{attribute 'linkalways'} 
{attribute 'no_explicit_call' := 'This FB is a CLASS and must be accessed using methods or properties'}
{attribute 'enable_dynamic_creation'}
FUNCTION_BLOCK Node_ContainerType_Vector_TcVnVector4_REAL EXTENDS Node
VAR
    out : _GUID;
END_VAR

METHOD PUBLIC  Clone : I_Node
VAR
	pNode : POINTER TO Node_ContainerType_Vector_TcVnVector4_REAL;
END_VAR
pNode := __NEW(Node_ContainerType_Vector_TcVnVector4_REAL);
Clone := pNode^;
END_METHOD

METHOD FB_init : BOOL
VAR_INPUT
	bInitRetains : BOOL; // if TRUE, the retain variables are initialized (warm start / cold start)
	bInCopyCode : BOOL;  // if TRUE, the instance afterwards gets moved into the copy code (online change)
END_VAR
AddOutput('out', out);
END_METHOD

METHOD PROTECTED OnExecute
out.Value := ContainerType_Vector_TcVnVector4_REAL;
END_METHOD

END_FUNCTION_BLOCK

(* stored: Version 1.1.0.1, ProductVersion 3.1.4026.17
   POU Node_ContainerType_Vector_TcVnVector4_REAL: Id {1a49ff89-4801-01e4-3b6e-50e6bc534b7d}, SpecialFunc None
   Folder Constructor: Id {15975e68-a1b3-0234-0d5b-a8292606f527}
   Method Clone: Id {49e122a4-5e02-0c86-3562-079590566fd4}
   Method FB_init: Id {036bfd92-b188-0f0f-2022-d54553331bc4}
   Method OnExecute: Id {dc8fec84-45d4-0b22-325c-bcd1fc4a3292} *)
